{attribute 'qualified_only'}
VAR_GLOBAL
END_VAR

(* stored: Version 1.1.0.1, ProductVersion 3.1.4022.7
   GVL GVL_07_Alarm_Servo_Motor_Shelf_Z: Id {a30e81d8-328e-47da-bb97-0becb409bb68} *)
